PROGRAM MAIN
VAR
END_VAR

END_PROGRAM

(* stored: Version 1.1.0.1
   POU MAIN: Id {b373c65c-8356-4dcc-8e42-53aa4067de3d} *)
